TYPE
    TcoSmartFunctionKitIO :
    STRUCT

        Response : TcoSmartFunctionKitResponseHw;
        Request : TcoSmartFunctionKitRequestHw;

    END_STRUCT
END_TYPE

(* stored: Version 1.1.0.1
   DUT TcoSmartFunctionKitIO: Id {a5bf0596-9aef-0ba4-1fa5-6ad077d52294} *)
